{attribute 'GeneratedUsingTerminal: EL1258-0010-0017'}
{attribute addProperty BoxType "EL1258-0010-0017"}
{attribute addProperty Id "Input_event_state_1BOOL1"}
{attribute addProperty CRC "271392008"}
{attribute addProperty Size "1"}
TYPE Inputs_102D1D08 :
STRUCT
	{attribute addProperty Name "Input_event_state_1"}
	Input_event_state_1 : BOOL;
END_STRUCT
END_TYPE

(* stored: Version 1.2.0.0, ProductVersion 3.1.4024.9
   DUT Inputs_102D1D08: Id {107cb7d5-8019-47d3-bdd9-c7ac2c7d721c} *)
